{attribute 'qualified_only'}
VAR_GLOBAL
  Com : ZCom;
END_VAR
VAR_GLOBAL PERSISTENT
  Data : ZData;
END_VAR

(* stored: Version 1.1.0.1
   GVL ZGlobal: Id {b4eba832-c0eb-48b5-a5ff-c23687a5a675} *)
